GLOBALCONSTANTS ISO_NETEVENT_e (* Global constants for network management event types *)
  (* Standard: 61499-1 *)
  (* Version 1.0, 2025-10-18, franz *)
  PACKAGE isobus::pgn;
  VAR_GLOBAL CONSTANT
    Isonet_MemberActive : USINT := 0;
    Isonet_MemberAddressConflict : USINT := 1; (* < There is a new member on network (intern or extern) *)
    Isonet_MemberInactive : USINT := 2; (* < Network member has lost address conflict *)
    Isonet_MemberNewAddress : USINT := 3; (* < Member stopped or commanded address *)
    Isonet_MemberAddressViolation : USINT := 4; (* < Address claimed after SA conflict *)
    Isonet_MemberAdd : USINT := 5; (* < Address violation: internal SA conflicts with SA from extern msg *)
    Isonet_MemberRemove : USINT := 6; (* < Core/base internal: Add(ed) CF to list *)
    Isonet_HsiActive : USINT := 7; (* Conditional constants from C-Code: #if defined (CCI_HSI) *)
    Isonet_HsiInactive : USINT := 8;
    Isonet_Last : USINT := 9; (* End of conditional block *)
  END_VAR
END_GLOBALCONSTANTS
